(* IEC 61131-3 sources: RL_MAR/experiments/comparison/autoplc/results/gpt-4o_20260511_211137/med_73, 1 file *)

(* ---- med_73_1.st ---- *)
FUNCTION_BLOCK RoboticWeldingSystem
    VAR_INPUT
        RobotArm1Ready : BOOL; (* Input for robot arm 1 ready status *)
        RobotArm2Ready : BOOL; (* Input for robot arm 2 ready status *)
        WeldingGunReady : BOOL; (* Input for welding gun ready status *)
        StartButton : BOOL; (* Input for start button press *)
        StopButton : BOOL; (* Input for stop button press *)
    END_VAR

    VAR_OUTPUT
        WeldingTrigger : BOOL; (* Output to trigger welding *)
        WeldingComplete : BOOL; (* Output indicating welding completion *)
    END_VAR

    VAR
        IsWelding : BOOL; (* Internal flag to track welding state *)
    END_VAR

    (* Initialization *)
    WeldingTrigger := FALSE;
    WeldingComplete := TRUE;
    IsWelding := FALSE;

    (* Main Control Logic *)
    IF StopButton THEN
        (* Safety Stop State *)
        WeldingTrigger := FALSE;
        WeldingComplete := TRUE;
        IsWelding := FALSE;
    ELSE
        IF RobotArm1Ready AND RobotArm2Ready AND WeldingGunReady AND StartButton THEN
            (* Welding State *)
            WeldingTrigger := TRUE;
            WeldingComplete := FALSE;
            IsWelding := TRUE;
        ELSE
            (* Idle State *)
            WeldingTrigger := FALSE;
            WeldingComplete := TRUE;
            IsWelding := FALSE;
        END_IF;
    END_IF;
END_FUNCTION_BLOCK
